ABB RobotStudio station: VRM_project_Cervenka.rspag

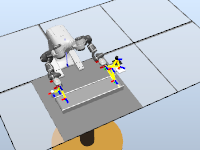
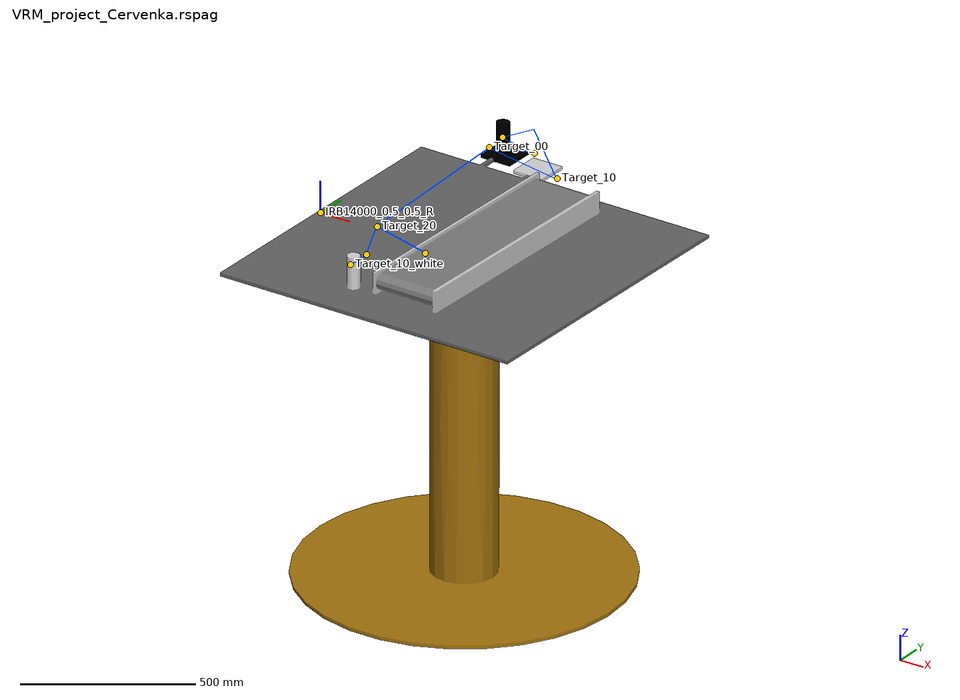
[picture v1: parts stored in the station drawn from their meshes, with robot base, taught points and paths (robot models come from the ABB library and are not in the file)]
--- station ---
Station Solution9 (saved by RobotStudio 21.4.9700.0)
Controller IRB14000
  mechanical unit ROB_R: IRB14000_0.5_0.5_R, 6 joints, base frame (0, 0, 0) mm
  mechanical unit ROB_R_7: IRB14000_0.5_0.5_R, 1 joints, base frame (0, 0, 0) mm
  mechanical unit ROB_L: IRB14000_0.5_0.5_L, 6 joints, base frame (0, 0, 0) mm
  mechanical unit ROB_L_7: IRB14000_0.5_0.5_L, 1 joints, base frame (0, 0, 0) mm
Layout (positions relative to the parent item):
  - IRB14000_0.5_0.5 [mechanism, from Robots\IRB14000_0.5_0.5__02.rslib] at (0, 0, 0) mm
  - IRB14000_0.5_0.5_R [mechanism, from Robots\IRB14000_0.5_0.5__02.rslib] at (0, 0, 0) mm; joint values [1.0732, -2.4606, -1.1122, 0.6063, 0.3644, 0.2549, 1.602] (rad or m)
  - IRB14000_0.5_0.5_L [mechanism, from Robots\IRB14000_0.5_0.5__02.rslib] at (0, 0, 0) mm; joint values [-0.8605, -2.3481, 1.1336, 0.3254, -0.2308, 0.5899, 1.1687] (rad or m)
  - Table [part], size 1000 x 1000 x 10 mm
  - Smart_Gripper_Servo_Fingers_2 [mechanism, from Tools\ABB_Smart_Gripper_Servo_Fingers.rslib] at (270.01, -267.25, 170.69) mm, rotated rx -90 ry 0 rz -90 deg; joint values [0.025] (rad or m)
  - Smart_Gripper_Servo_Fingers_3 [mechanism, from Tools\ABB_Smart_Gripper_Servo_Fingers.rslib] at (215.91, 366.18, 153.52) mm, rotated rx -90 ry 0 rz -90 deg; joint values [0.025] (rad or m)
  - Thing_White [part] at (215.38, 41.77, 1.05) mm, size 40 x 39.9 x 100 mm
  - Attacher_white [smart component, from Components\Attacher.rslib]
      properties: Parent=Smart_Gripper_Servo_Fingers_2; Flange=0; Child=Thing_White; Mount=false; Offset=[0 0 0]; Orientation=[0 0 0]
  - Detacher_white [smart component, from Components\Detacher.rslib]
      properties: Child=Thing_White; KeepPosition=true
  - LinearMover_white [smart component, from Components\LinearMover.rslib]
      properties: Object=Thing_White; Direction=[0 0.001 0]; Speed=0.1; Reference=Global; ReferenceObject=(none)
  - LineSensor [smart component, from Components\LineSensor.rslib]
      properties: Start=[0.446335 0.372458 0.08392]; End=[0.659285 0.381354 0.083895]; Radius=0; SensedPart=(none); SensedPoint=[0 0 0]
    - _sensorPart_ [part], size 212.9 x 8.9 x 0 mm
  - Positioner [smart component, from Components\Positioner.rslib]
      properties: Object=Thing_White; Position=[0.215378 0.041769 0.001054]; Orientation=[0 0 0]; Reference=Global; ReferenceObject=(none)
  - Attacher_2_white [smart component, from Components\Attacher.rslib] at (318.13, 59.56, 93.72) mm, rotated rx 0 ry 0 rz 72.88 deg
      properties: Parent=Smart_Gripper_Servo_Fingers_3; Flange=0; Child=Thing_White; Mount=false; Offset=[0 0 0]; Orientation=[0 0 0]
  - Detacher_2_white [smart component, from Components\Detacher.rslib]
      properties: Child=Thing_White; KeepPosition=true
  - PoseMover_R [smart component, from Components\PoseMover.rslib] at (476.57, -525.07, 0) mm
      properties: Mechanism=Smart_Gripper_Servo_Fingers_2; Pose=1; Duration=1
  - PoseMover_R [smart component, from Components\PoseMover.rslib]
      properties: Mechanism=Smart_Gripper_Servo_Fingers_2; Pose=2; Duration=1
  - PoseMover_L [smart component, from Components\PoseMover.rslib] at (370.45, -539.65, 0) mm
      properties: Mechanism=Smart_Gripper_Servo_Fingers_3; Pose=2; Duration=1
  - PoseMover_L [smart component, from Components\PoseMover.rslib] at (476.57, -525.07, 0) mm
      properties: Mechanism=Smart_Gripper_Servo_Fingers_3; Pose=1; Duration=1
  - Conveyor [part] at (-329.87, -300.54, -144.17) mm, size 228.6 x 802.4 x 70.3 mm
  - White_target [part] at (86.38, -71.44, -60.48) mm, size 100 x 100 x 10 mm
  - Black_target [part] at (-47.15, -40.78, -59.61) mm, size 100 x 100 x 10 mm
  - Thing_Black [part] at (-210.85, 614.86, -0.2) mm, rotated rx 0 ry 0 rz 67.12 deg, size 40 x 39.9 x 100 mm
  - Positioner_2 [smart component, from Components\Positioner.rslib]
      properties: Object=Thing_Black; Position=[0.215378 0.117 0.001054]; Orientation=[0 0 0]; Reference=Global; ReferenceObject=(none)
  - Part_2 [part] at (0, 0, -1007.26) mm, size 200 x 200 x 1000 mm
  - Part_3 [part], size 1000 x 994.5 x 10 mm
  - LinearMover_black [smart component, from Components\LinearMover.rslib]
      properties: Object=Thing_Black; Direction=[0 0.001 0]; Speed=0.1; Reference=Global; ReferenceObject=(none)
  - Part_4 [part] at (-191.96, -38.8, -4.88) mm, size 10 x 100 x 10 mm
  - Part_5 [part] at (-44.2, -69.14, -4.65) mm, size 10 x 100 x 10 mm
  - Attacher_black [smart component, from Components\Attacher.rslib]
      properties: Parent=Smart_Gripper_Servo_Fingers_2; Flange=0; Child=Thing_Black; Mount=false; Offset=[0 0 0]; Orientation=[0 0 0]
  - Attacher_2_black [smart component, from Components\Attacher.rslib]
      properties: Parent=Smart_Gripper_Servo_Fingers_3; Flange=0; Child=Thing_Black; Mount=false; Offset=[0 0 0]; Orientation=[0 0 0]
  - Detacher_black [smart component, from Components\Detacher.rslib]
      properties: Child=Thing_Black; KeepPosition=true
  - Detacher_2_black [smart component, from Components\Detacher.rslib]
      properties: Child=Thing_Black; KeepPosition=true
  - LogicGate_2 [smart component, from Components\LogicGate.rslib]
      properties: Operator=AND; Delay=0
  - LogicGate_3 [smart component, from Components\LogicGate.rslib]
      properties: Operator=AND; Delay=0
  - LogicGate_4 [smart component, from Components\LogicGate.rslib]
      properties: Operator=NOT; Delay=0
  - LogicGate_5 [smart component, from Components\LogicGate.rslib]
      properties: Operator=AND; Delay=0
  - LogicGate_6 [smart component, from Components\LogicGate.rslib]
      properties: Operator=AND; Delay=0
  - LogicGate_7 [smart component, from Components\LogicGate.rslib]
      properties: Operator=AND; Delay=0
  - LogicGate_8 [smart component, from Components\LogicGate.rslib]
      properties: Operator=AND; Delay=0
Attachment: Smart_Gripper_Servo_Fingers_2 is attached to IRB14000_0.5_0.5_R / Link7
Attachment: Smart_Gripper_Servo_Fingers_3 is attached to IRB14000_0.5_0.5_L / Link7
Attachment: LinearMover_white is attached to Table
Attachment: Attacher_2_white is attached to IRB14000_0.5_0.5_L / Link7
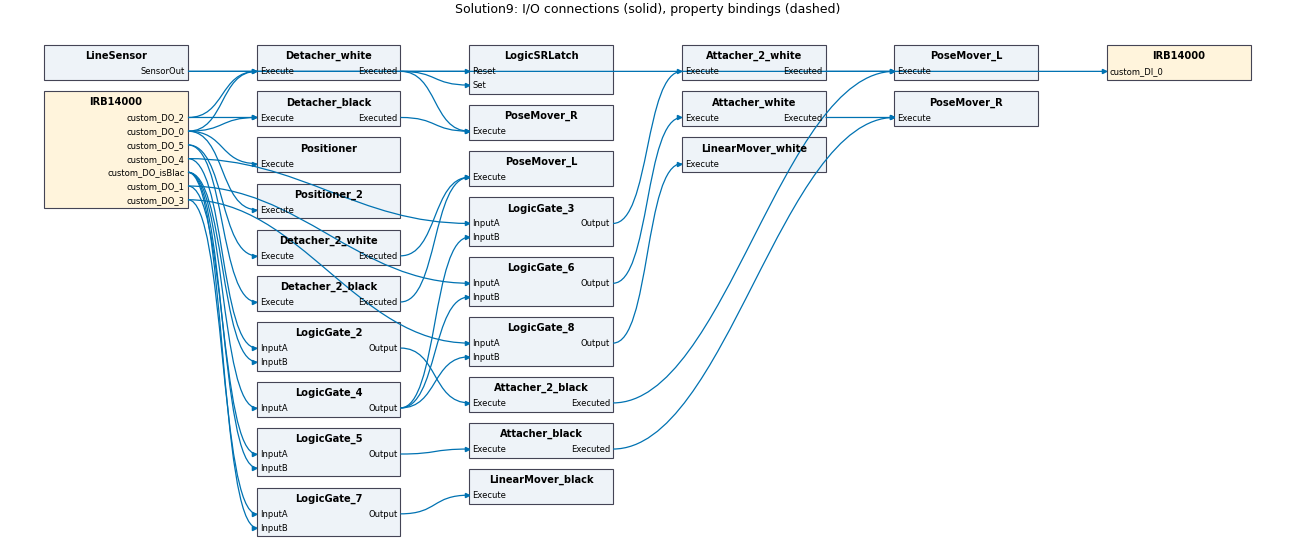
Station logic (signal -> signal, property => property):
  LineSensor.SensorOut -> LogicSRLatch.Reset
  IRB14000.custom_DO_2 -> Detacher_white.Execute
  Detacher_white.Executed -> LogicSRLatch.Set
  IRB14000.custom_DO_0 -> Positioner.Execute
  IRB14000.custom_DO_0 -> Detacher_white.Execute
  LineSensor.SensorOut -> IRB14000.custom_DI_0
  IRB14000.custom_DO_5 -> Detacher_2_white.Execute
  Attacher_white.Executed -> PoseMover_R.Execute
  Detacher_white.Executed -> PoseMover_R.Execute
  Attacher_2_white.Executed -> PoseMover_L.Execute
  Detacher_2_white.Executed -> PoseMover_L.Execute
  IRB14000.custom_DO_0 -> Positioner_2.Execute
  IRB14000.custom_DO_5 -> Detacher_2_black.Execute
  IRB14000.custom_DO_2 -> Detacher_black.Execute
  IRB14000.custom_DO_0 -> Detacher_black.Execute
  Detacher_2_black.Executed -> PoseMover_L.Execute
  IRB14000.custom_DO_4 -> LogicGate_2.InputA
  LogicGate_2.Output -> Attacher_2_black.Execute
  Attacher_2_black.Executed -> PoseMover_L.Execute
  IRB14000.custom_DO_isBlack -> LogicGate_2.InputB
  IRB14000.custom_DO_4 -> LogicGate_3.InputA
  IRB14000.custom_DO_isBlack -> LogicGate_4.InputA
  LogicGate_4.Output -> LogicGate_3.InputB
  LogicGate_3.Output -> Attacher_2_white.Execute
  IRB14000.custom_DO_1 -> LogicGate_5.InputA
  LogicGate_5.Output -> Attacher_black.Execute
  IRB14000.custom_DO_isBlack -> LogicGate_5.InputB
  IRB14000.custom_DO_1 -> LogicGate_6.InputA
  LogicGate_4.Output -> LogicGate_6.InputB
  LogicGate_6.Output -> Attacher_white.Execute
  Attacher_black.Executed -> PoseMover_R.Execute
  Detacher_black.Executed -> PoseMover_R.Execute
  LogicGate_7.Output -> LinearMover_black.Execute
  IRB14000.custom_DO_3 -> LogicGate_7.InputA
  IRB14000.custom_DO_3 -> LogicGate_8.InputA
  LogicGate_4.Output -> LogicGate_8.InputB
  LogicGate_8.Output -> LinearMover_white.Execute
  IRB14000.custom_DO_isBlack -> LogicGate_7.InputB

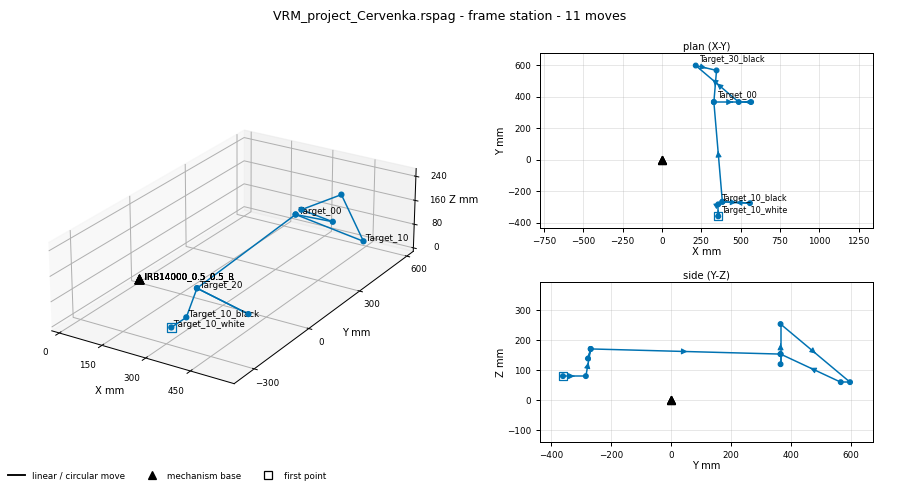
[picture p0: tool path of VRM_project_Cervenka.rspag in frame station, 11 of 11 moves have a stored position in this frame; points joined in program order, loops and branches not executed]
--- Backups/IRB14000/RAPID/TASK1/PROGMOD/CalibData.mod ---
MODULE CalibData
    PERS tooldata Servo:=[TRUE,[[0,0,114.2],[1,0,0,0]],[0.215,[8.7,12.3,49.2],[1,0,0,0],0.00021,0.00024,0.00009]];
    PERS tooldata Tooldata_1:=[TRUE,[[0,0,114.2],[1,0,0,0]],[0.215,[8.7,12.3,49.2],[1,0,0,0],0.00021,0.00024,0.00009]];
ENDMODULE

--- Backups/IRB14000/RAPID/TASK1/PROGMOD/Module1.mod ---
MODULE Module1
        CONST robtarget Target_10:=[[357.994922696,-359.830403815,79.958971591],[0.5,-0.5,0.5,-0.5],[1,0,1,4],[-101.964426493,9E+09,9E+09,9E+09,9E+09,9E+09]];
    CONST robtarget Target_20:=[[384.208016924,-267.247186969,170.693355338],[0.5,-0.5,0.5,-0.5],[1,0,1,4],[-101.964426493,9E+09,9E+09,9E+09,9E+09,9E+09]];
    CONST robtarget Target_30:=[[559.354511697,-276.222648897,138.649291138],[0.5,-0.5,0.5,-0.5],[1,0,1,4],[-101.964426493,9E+09,9E+09,9E+09,9E+09,9E+09]];
    CONST robtarget Target_40:=[[294.263,78.1,59.804],[0.704416026,-0.704416026,-0.061628417,0.061628417],[0,0,0,0],[-101.96443162,9E+09,9E+09,9E+09,9E+09,9E+09]];
    CONST robtarget Target_10_white:=[[357.994922696,-359.830403815,79.958971591],[0.5,-0.5,0.5,-0.5],[1,0,1,4],[-101.964426493,9E+09,9E+09,9E+09,9E+09,9E+09]];
    CONST robtarget Target_10_black:=[[357.994945982,-283.42680044,79.959185144],[0.500001497,-0.500001497,0.499998503,-0.499998503],[1,0,1,4],[-101.964429355,9E+09,9E+09,9E+09,9E+09,9E+09]];
!***********************************************************
    !
    ! Module:  Module1
    !
    ! Description:
    !   <Insert description here>
    !
    ! Author: suiti
    !
    ! Version: 1.0
    !
    !***********************************************************


    !***********************************************************
    !
    ! Procedure main
    !
    !   This is the entry point of your program
    !
    !***********************************************************
    PROC main()
            SetDO custom_DO_isBlack, custom_DI_isBlack; ! set D0 is black to value of DI is black
            Path_10;
    ENDPROC
    PROC Path_10()
        PulseDO custom_DO_0; !reset
        IF custom_DI_isBlack = 0 THEN
            MoveL Target_10_white,v1000,fine,Tooldata_1\WObj:=wobj0;
        ELSE
            MoveL Target_10_black,v1000,fine,Tooldata_1\WObj:=wobj0;
        ENDIF
        PulseDO custom_DO_1; !attach
        WaitTime \InPos, 1;
        MoveL Target_20,v1000,fine,Tooldata_1\WObj:=wobj0;
        MoveL Target_30,v1000,fine,Tooldata_1\WObj:=wobj0;
        PulseDO custom_DO_2; !detach
        WaitTime 1;
        MoveL Target_20,v1000,fine,Tooldata_1\WObj:=wobj0;
        SetDO custom_DO_3, 1; ! run conveyor
        WaitUntil custom_DI_0 = 1; !sensor
        !off conveyor
        SetDO custom_DO_3,0;

    ENDPROC
ENDMODULE

--- Backups/IRB14000/RAPID/TASK2/PROGMOD/CalibData.mod ---
MODULE CalibData
    PERS tooldata Servo:=[TRUE,[[0,0,114.2],[1,0,0,0]],[0.215,[8.7,12.3,49.2],[1,0,0,0],0.00021,0.00024,0.00009]];
ENDMODULE

--- Backups/IRB14000/RAPID/TASK2/PROGMOD/Module1.mod ---
MODULE Module1
        CONST robtarget Target_00:=[[330.112611472,366.177,153.522304411],[0.5,-0.5,0.5,-0.5],[-1,0,1,4],[101.964427132,9E+09,9E+09,9E+09,9E+09,9E+09]];
    CONST robtarget Target_10:=[[566.737,366.177,119.744],[0.5,-0.5,0.5,-0.5],[-1,0,0,4],[101.964427132,9E+09,9E+09,9E+09,9E+09,9E+09]];
    CONST robtarget Target_20:=[[487.799658063,366.177,253.748829607],[0.5,-0.5,0.5,-0.5],[-1,1,0,4],[101.964427132,9E+09,9E+09,9E+09,9E+09,9E+09]];
    CONST robtarget Target_30:=[[296.557038398,78.806214933,59.803604774],[0.105248534,-0.105248534,0.69923011,-0.69923011],[-1,1,0,4],[101.964427132,9E+09,9E+09,9E+09,9E+09,9E+09]];
    CONST robtarget Target_30_black:=[[214.91709963,597.987319612,59.803604774],[0.693058493,-0.693058493,0.140249511,-0.140249511],[-1,1,0,4],[101.964427132,9E+09,9E+09,9E+09,9E+09,9E+09]];
    CONST robtarget Target_30_white:=[[347.120135833,566.991935769,59.803604774],[0.633977721,-0.633977721,0.313164891,-0.313164891],[-1,1,0,4],[101.964427132,9E+09,9E+09,9E+09,9E+09,9E+09]];

    !PERS bool isBlack := FALSE;
!***********************************************************
    !
    ! Module:  Module1
    !
    ! Description:
    !   <Insert description here>
    !
    ! Author: suiti
    !
    ! Version: 1.0
    !
    !***********************************************************


    !***********************************************************
    !
    ! Procedure main
    !
    !   This is the entry point of your program
    !
    !***********************************************************
    PROC main()
        Path_10;
    ENDPROC
    PROC Path_10() !path for white
        WaitUntil custom_DI_0 = 1 AND custom_DO_3 = 0; !signal from 1st robot and sensor
        MoveL Target_00,v1000,z100,Servo\WObj:=wobj0;
        MoveL Target_10,v1000,fine,Servo\WObj:=wobj0;
        WaitTime \InPos, 1;
        PulseDO custom_DO_4; !attach
        MoveL Target_20,v1000,fine,Servo\WObj:=wobj0;
        IF custom_DI_isBlack = 1 THEN
            MoveL Target_30_black,v1000,fine,Servo\WObj:=wobj0;
        ELSE
            MoveL Target_30_white,v1000,fine,Servo\WObj:=wobj0;
        ENDIF
        PulseDO custom_DO_5;
        MoveL Target_00, v1000, fine, Servo\WObj:=wobj0;
    ENDPROC
ENDMODULE

--- Backups/IRB14000/SYSPAR/EIO.cfg ---
EIO:CFG_1.0:6:1::
#
SYSSIG_IN:

      -Signal "Collision_Avoidance" -Action "CollAvoidance"
#
INDUSTRIAL_NETWORK:

      -Name "EtherNetIP" -Connection "Private Network"\
      -Label "EtherNet/IP Adapter Network"

      -Name "DeviceNet" -Label "DeviceNet Master/Slave Network" -Address "2"
#
EIO_CROSS:

      -Name "Cross_Signal_Lamp" -Res "Signal_Lamp" -Act1 "DRV1BRAKE"
#
EIO_SIGNAL_SAFELEVEL:

      -Name "FlangePowerSafeLevel" -ActionWhenStartup "Last"
#
DEVICENET_DEVICE:

      -Name "D652_10" -VendorName "ABB Robotics" -ProductName "24 VDC Unit"\
      -Address 10 -ProductCode 26 -DeviceType 7 -ConnectionType "COS"\
      -OutputSize 2 -InputSize 2
#
DEVICENET_INTERNAL_DEVICE:

      -Name "DN_Internal_Device" -VendorName "ABB Robotics"\
      -ProductName "DeviceNet Internal Slave Device"
#
ETHERNETIP_INTERNAL_DEVICE:

      -Name "EN_Internal_Device" -VendorName "ABB Robotics"\
      -ProductName "EtherNet/IP Internal Adapter Device"
#
EIO_SIGNAL:

      -Name "custom_DI_0" -SignalType "DI" -Device "D652_10" -DeviceMap "0"

      -Name "custom_DI_1" -SignalType "DI" -Device "D652_10" -DeviceMap "1"

      -Name "custom_DI_2" -SignalType "DI" -Device "D652_10" -DeviceMap "2"

      -Name "custom_DI_3" -SignalType "DI" -Device "D652_10" -DeviceMap "3"

      -Name "custom_DI_4" -SignalType "DI" -Device "D652_10" -DeviceMap "4"

      -Name "custom_DI_5" -SignalType "DI" -Device "D652_10" -DeviceMap "5"

      -Name "custom_DI_6" -SignalType "DI" -Device "D652_10" -DeviceMap "6"

      -Name "custom_DI_isBlack" -SignalType "DI" -Device "D652_10"\
      -DeviceMap "7"

      -Name "custom_DO_0" -SignalType "DO" -Device "D652_10" -DeviceMap "0"

      -Name "custom_DO_1" -SignalType "DO" -Device "D652_10" -DeviceMap "1"

      -Name "custom_DO_2" -SignalType "DO" -Device "D652_10" -DeviceMap "2"

      -Name "custom_DO_3" -SignalType "DO" -Device "D652_10" -DeviceMap "3"

      -Name "custom_DO_4" -SignalType "DO" -Device "D652_10" -DeviceMap "4"

      -Name "custom_DO_5" -SignalType "DO" -Device "D652_10" -DeviceMap "5"

      -Name "custom_DO_6" -SignalType "DO" -Device "D652_10" -DeviceMap "6"

      -Name "custom_DO_isBlack" -SignalType "DO" -Device "D652_10"\
      -DeviceMap "7"

      -Name "hall_sensor_joint_1" -SignalType "DI" -Device "D652_10"\
      -DeviceMap "8"

      -Name "hall_sensor_joint_2" -SignalType "DI" -Device "D652_10"\
      -DeviceMap "9"

      -Name "hall_sensor_joint_3" -SignalType "DI" -Device "D652_10"\
      -DeviceMap "11"

      -Name "hall_sensor_joint_4" -SignalType "DI" -Device "D652_10"\
      -DeviceMap "12"

      -Name "hall_sensor_joint_5" -SignalType "DI" -Device "D652_10"\
      -DeviceMap "13"

      -Name "hall_sensor_joint_6" -SignalType "DI" -Device "D652_10"\
      -DeviceMap "14"

      -Name "hall_sensor_joint_7" -SignalType "DI" -Device "D652_10"\
      -DeviceMap "10"

      -Name "hall_sensor_24V_ROB_R" -SignalType "DO" -Device "D652_10"\
      -DeviceMap "8"

      -Name "hall_sensor_24V_ROB_L" -SignalType "DO" -Device "D652_10"\
      -DeviceMap "9"

      -Name "flange_24V_ROB_R" -SignalType "DO" -Device "D652_10"\
      -DeviceMap "10" -SafeLevel "FlangePowerSafeLevel"

      -Name "flange_24V_ROB_L" -SignalType "DO" -Device "D652_10"\
      -DeviceMap "11" -SafeLevel "FlangePowerSafeLevel"

      -Name "Signal_Lamp" -SignalType "DO" -Device "D652_10" -DeviceMap "12"

      -Name "Collision_Avoidance" -SignalType "DO" -Access "All" -Default 1
